FUNCTION Convert_DATE_TO_DT : Hresult
VAR_INPUT
	in : DATE;
	out : REFERENCE TO DT;
END_VAR
VAR
	converted : DT;
END_VAR
VAR CONSTANT
	INCOMPATIBLE : HRESULT := 16#9811070E;
END_VAR

converted := DATE_TO_DT(in);

IF (DT_TO_DATE(converted) <> in) THEN
	Convert_DATE_TO_DT := INCOMPATIBLE;
	RETURN;
END_IF

out := converted;

END_FUNCTION

(* stored: Version 1.1.0.1, ProductVersion 3.1.4024.12
   POU Convert_DATE_TO_DT: Id {2c36ab1a-e781-4750-b44b-96c3c64fc385}, SpecialFunc None *)
